INTERFACE I_Reset

METHOD Reset
VAR_INPUT
	Execute : BOOL;
END_VAR
END_METHOD

PROPERTY ResetBusy : BOOL
GET
END_GET
END_PROPERTY

PROPERTY ResetDone : BOOL
GET
END_GET
END_PROPERTY

PROPERTY ResetError : BOOL
GET
END_GET
END_PROPERTY

PROPERTY ResetErrorID : UDINT
GET
END_GET
END_PROPERTY

END_INTERFACE

(* stored: Version 1.1.0.1
   Itf I_Reset: Id {b13e0a07-13fe-4130-92d2-b67a6bf512d3}
   Method Reset: Id {6de39cad-1884-4ec7-b494-38b114cd7658}
   Property ResetBusy: Id {0dcd0461-4313-48f9-8cd0-fb4c21feef7d}
   Get Get: Id {60e12a27-7f75-4317-b2bc-2d250342c39c}
   Property ResetDone: Id {bb784cbf-17a8-432f-aadf-22fcb5fecc6c}
   Get Get: Id {f83b19e6-00dd-4fa2-8d16-a92fd4d26631}
   Property ResetError: Id {df9aa5b8-56fc-4693-865f-0277cf76b958}
   Get Get: Id {b0a6c8d5-7534-4098-9b97-c37ee815f05f}
   Property ResetErrorID: Id {7fd91d91-4ae3-41d2-a2a6-3db4fead9dd5}
   Get Get: Id {7849cabf-22f5-4195-800f-ea3857cd3a2b} *)
